// TIA Portal V14 SP1 export
// export: Created 2019-05-16T13:33:21.7383868Z, ExportSetting WithDefaults, WithReadOnly, DisplayName Totally Integrated Automation Portal, DisplayVersion V14 SP1 Update 6, DisplayName TIA Portal Openness, DisplayVersion V14 SP1 Update 6, DisplayName STEP 7 Professional, DisplayVersion V14 SP1 Update 6, DisplayName WinCC Professional, DisplayVersion V14 SP1 Update 6
FUNCTION_BLOCK "408М_Компрессор"   // FB2026, LAD
{ S7_Optimized_Access := 'FALSE' }
VERSION : 0.1
// stored: AutoNumber false, CodeModifiedDate 2019-03-26T07:08:54.9645568Z, CompileDate 2019-03-26T07:08:54.9928771Z, CreationDate 2019-02-26T05:18:41.6523018Z, InterfaceModifiedDate 2019-03-06T13:28:02.3471097Z, IsConsistent true, IsIECCheckEnabled false, IsKnowHowProtected false, ISMultiInstanceCapable true, IsWriteProtected false, LibraryConformanceStatus Warning: The object contains access to global data blocks. Warning: The block contains direct access to inputs, outputs, bit memories, indirect access to the registry or indirect access to external memory areas that are unknown at the time of compilation., ModifiedDate 2019-03-26T07:08:54.9645568Z, ParameterModified 2019-01-09T12:59:30.7163193Z, StructureModified 2019-03-06T13:28:02.3471097Z, UDAEnableTagReadback false
   VAR DB_SPECIFIC
      HMI : Struct
         CMD : Struct
            Start : Bool;   // Команда старта вибратора
            Stop : Bool;   // Команда останова вибратора
            Spare_2 : Bool;
            Spare_3 : Bool;
            Spare_4 : Bool;
            Spare_5 : Bool;
            Manual : Bool;
            Reset_Error : Bool;   // Сброс ошибок
         END_STRUCT;
         DATA : Struct
            StatusWord : Word;
            CntFbkTime : DInt := 4;   // Время контроля включения реле
            TimeDelay_SP : DInt := 2;   // Задержка срабатывания датчика давления
            Rot_Off_Time : Int;   // Обратный отсчет времени задержки запуска
            Line_Pressure_OK : Bool;   // Датчик давления компрессора ОК / Датчик давления в линии компрессора ОК
            Compressor_Pressure_OK : Bool;   // Датчик давления компрессора ОК
            Spare_7 : Bool;
            Spare_8 : Bool;
            Spare_9 : Bool;
            Spare_10 : Bool;
            Spare_11 : Bool;
            Spare_6 : Bool;
            Line_Presure : Real;   // Значение давления в линии
         END_STRUCT;
      END_STRUCT;
   END_VAR
   VAR
      One_Motor : "OneMotorManag";
      TOF : TOF;
      TOF_1 : TOF;
      TP : TP;
   END_VAR
   VAR DB_SPECIFIC
      CntFbkTime : Time;
      TimeDelay_SP : Time;
      StopTime : Time;   // Время остановки мотора компрессора
      Line_Presure : Real;   // Значение давления в линии
      Sensor_SP_OK : Bool;   // Датчик давления OK
      ResetErr : Bool;   // Сброс ошибок / Dumping of errors of the control package
      General_cond_OK : Bool;   // Готовность электрических систем / Conditions of permission of operation of the mechanism are not satisfied
      ManCmd_StartMov : Bool;   // Старт вращения в ручном режиме / Existence of command for rotation of the motor in manual
      ManCmd_StopMov : Bool;   // Стоп вращения в ручном режиме / Existence of command for a stop of rotation of the motor in manual
      AutoCmd_StartMov : Bool;   // Старт вращения в автоматическом режиме / Existence of command for rotation of the motor in the automatic
      AutoCmd_StopMov : Bool;   // Стоп вращения в автоматическом режиме / Existence of command for a stop of rotation of the motor in the automatic
   END_VAR
   VAR_TEMP
      FErr : Bool;   // Command 1 on operation of the mechanism in the automatic mode
      Temp_DINT : DInt;
   END_VAR
   VAR_TEMP   // added for the SCL form of the ladder/FBD networks
      _w1 : Bool;
      _w2 : Bool;
   END_VAR
BEGIN

REGION Network 2: Сброс ошибок
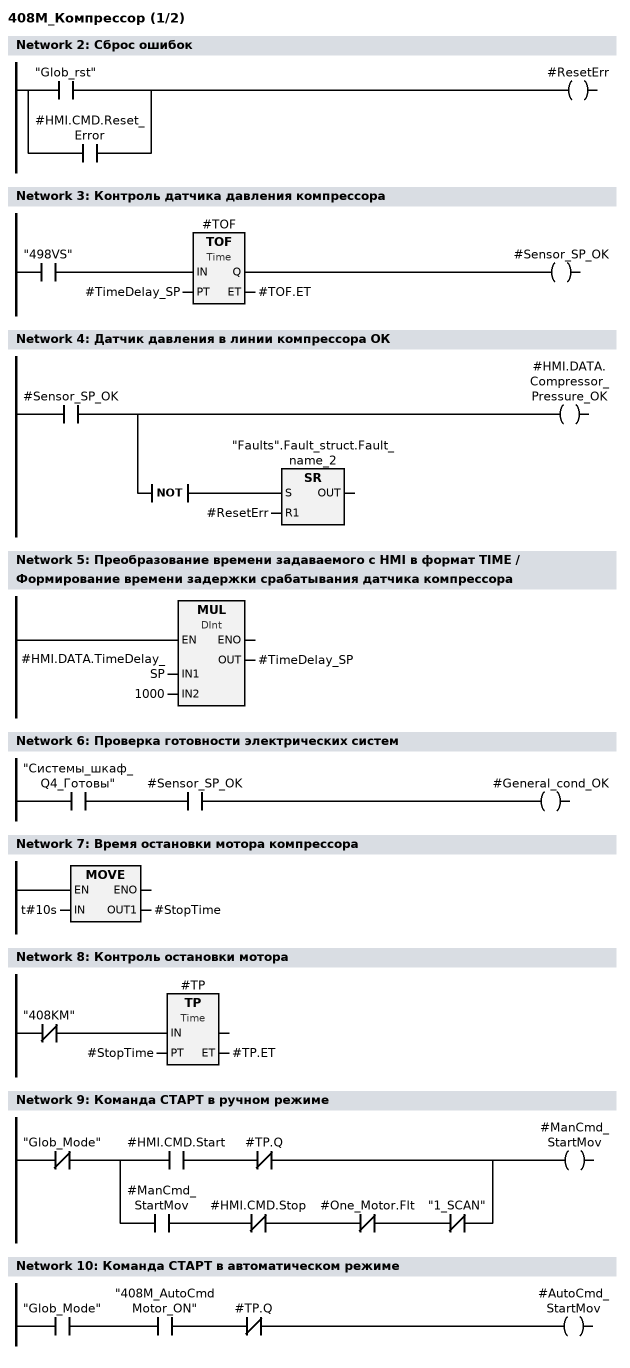
   RUNG wire#powerrail
      Contact( "Glob_rst" )
      wire#w1
      Coil( #ResetErr )
   END_RUNG
   RUNG wire#powerrail
      Contact( #HMI.CMD.Reset_Error )
   END_RUNG wire#w1
   // the same network as SCL:
   #ResetErr := "Glob_rst" OR #HMI.CMD.Reset_Error;
END_REGION

REGION Network 3: Контроль датчика давления компрессора
   RUNG wire#powerrail
      Contact( "498VS" )
      { S7_Templates := "time_type := Time" } #TOF.TOF(pt := #TimeDelay_SP, et => #TOF.ET)
      Coil( #Sensor_SP_OK )
   END_RUNG
   // the same network as SCL:
   #TOF.TOF(IN := "498VS", PT := #TimeDelay_SP, ET => #TOF.ET);
   #Sensor_SP_OK := #TOF.Q;
END_REGION

REGION Network 4: Датчик давления в линии компрессора ОК
   RUNG wire#powerrail
      Contact( #Sensor_SP_OK )
      wire#w1
      Coil( #HMI.DATA.Compressor_Pressure_OK )
   END_RUNG
   RUNG wire#w1
      Not()
      S_SR(operand := "Faults".Fault_struct.Fault_name_2, r1 := #ResetErr)
   END_RUNG
   // the same network as SCL:
   #HMI.DATA.Compressor_Pressure_OK := #Sensor_SP_OK;
   IF NOT #Sensor_SP_OK THEN
       "Faults".Fault_struct.Fault_name_2 := TRUE;   // SR flip-flop
   END_IF;
   IF #ResetErr THEN "Faults".Fault_struct.Fault_name_2 := FALSE; END_IF;
END_REGION

REGION Network 5: Преобразование времени задаваемого с HMI в формат TIME / Формирование времени задержки срабатывания датчика компрессора
   RUNG wire#powerrail
      { S7_Templates := "SrcType := DInt"; S7_GenerateENO := "TRUE" } Mul(in1 := #HMI.DATA.TimeDelay_SP, in2 := 1000, out => #TimeDelay_SP)
   END_RUNG
   // the same network as SCL:
   #TimeDelay_SP := #HMI.DATA.TimeDelay_SP * 1000;
END_REGION

REGION Network 6: Проверка готовности электрических систем
   RUNG wire#powerrail
      Contact( "Системы_шкаф_Q4_Готовы" )
      Contact( #Sensor_SP_OK )
      Coil( #General_cond_OK )
   END_RUNG
   // the same network as SCL:
   #General_cond_OK := "Системы_шкаф_Q4_Готовы" AND #Sensor_SP_OK;
END_REGION

REGION Network 7: Время остановки мотора компрессора
   RUNG wire#powerrail
      { S7_GenerateENO := "TRUE" } Move(in := t#10s, out1 => #StopTime)
   END_RUNG
   // the same network as SCL:
   #StopTime := t#10s;
END_REGION

REGION Network 8: Контроль остановки мотора
   RUNG wire#powerrail
      I_Contact( "408KM" )
      { S7_Templates := "time_type := Time" } #TP.TP(pt := #StopTime, et => #TP.ET)
   END_RUNG
   // the same network as SCL:
   #TP.TP(IN := NOT "408KM", PT := #StopTime, ET => #TP.ET);
END_REGION

REGION Network 9: Команда СТАРТ в ручном режиме
   RUNG wire#powerrail
      I_Contact( "Glob_Mode" )
      wire#w1
      Contact( #HMI.CMD.Start )
      I_Contact( #TP.Q )
      wire#w2
      Coil( #ManCmd_StartMov )
   END_RUNG
   RUNG wire#w1
      Contact( #ManCmd_StartMov )
      I_Contact( #HMI.CMD.Stop )
      I_Contact( #One_Motor.Flt )
      I_Contact( "1_SCAN" )
   END_RUNG wire#w2
   // the same network as SCL:
   #ManCmd_StartMov := NOT "Glob_Mode" AND ((#HMI.CMD.Start AND NOT #TP.Q) OR (#ManCmd_StartMov AND NOT #HMI.CMD.Stop AND NOT #One_Motor.Flt AND NOT "1_SCAN"));
END_REGION

REGION Network 10: Команда СТАРТ в автоматическом режиме
   RUNG wire#powerrail
      Contact( "Glob_Mode" )
      Contact( "408M_AutoCmdMotor_ON" )
      I_Contact( #TP.Q )
      Coil( #AutoCmd_StartMov )
   END_RUNG
   // the same network as SCL:
   #AutoCmd_StartMov := "Glob_Mode" AND "408M_AutoCmdMotor_ON" AND NOT #TP.Q;
END_REGION

REGION Network 11: Преобразование времени задаваемого с HMI в формат TIME
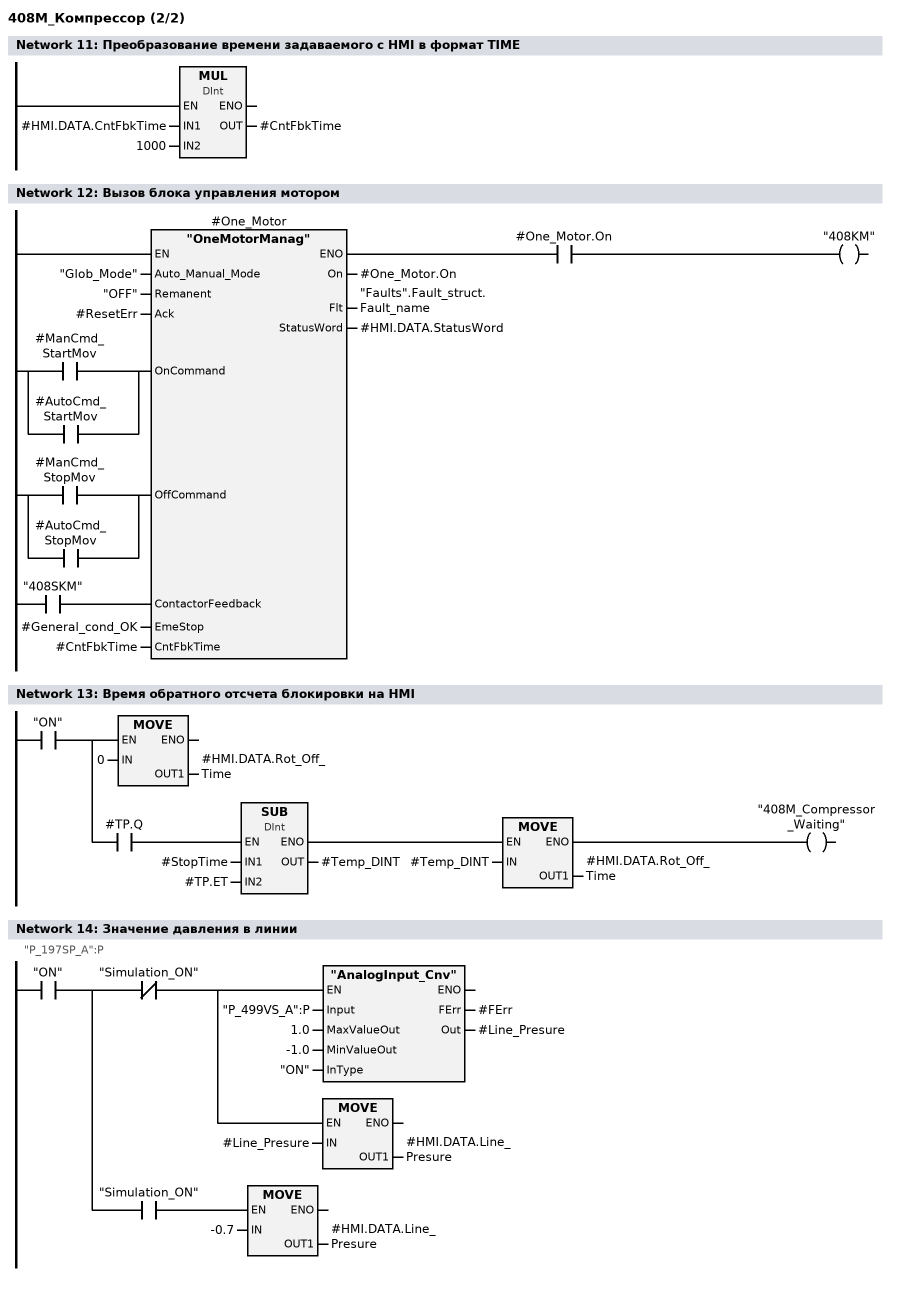
   RUNG wire#powerrail
      { S7_Templates := "SrcType := DInt"; S7_GenerateENO := "TRUE" } Mul(in1 := #HMI.DATA.CntFbkTime, in2 := 1000, out => #CntFbkTime)
   END_RUNG
   // the same network as SCL:
   #CntFbkTime := #HMI.DATA.CntFbkTime * 1000;
END_REGION

REGION Network 12: Вызов блока управления мотором
   RUNG wire#powerrail
      #One_Motor(OnCommand := wire#w1, OffCommand := wire#w2, ContactorFeedback := wire#w3, Auto_Manual_Mode := "Glob_Mode", Remanent := "OFF", Ack := #ResetErr, EmeStop := #General_cond_OK, CntFbkTime := #CntFbkTime, On => #One_Motor.On, Flt => "Faults".Fault_struct.Fault_name, StatusWord => #HMI.DATA.StatusWord)
      Contact( #One_Motor.On )
      Coil( "408KM" )
   END_RUNG
   RUNG wire#powerrail
      Contact( #ManCmd_StartMov )
   END_RUNG wire#w1
   RUNG wire#powerrail
      Contact( #AutoCmd_StartMov )
   END_RUNG wire#w1
   RUNG wire#powerrail
      Contact( #ManCmd_StopMov )
   END_RUNG wire#w2
   RUNG wire#powerrail
      Contact( #AutoCmd_StopMov )
   END_RUNG wire#w2
   RUNG wire#powerrail
      Contact( "408SKM" )
   END_RUNG wire#w3
   // the same network as SCL:
   #One_Motor(Auto_Manual_Mode := "Glob_Mode",   // "OneMotorManag"
              Remanent := "OFF",
              Ack := #ResetErr,
              OnCommand := #ManCmd_StartMov OR #AutoCmd_StartMov,
              OffCommand := #ManCmd_StopMov OR #AutoCmd_StopMov,
              ContactorFeedback := "408SKM",
              EmeStop := #General_cond_OK,
              CntFbkTime := #CntFbkTime,
              On => #One_Motor.On,
              Flt => "Faults".Fault_struct.Fault_name,
              StatusWord => #HMI.DATA.StatusWord,
              ENO => #_w1);
   "408KM" := #_w1 AND #One_Motor.On;
END_REGION

REGION Network 13: Время обратного отсчета блокировки на HMI
   RUNG wire#powerrail
      Contact( "ON" )
      wire#w1
      { S7_GenerateENO := "TRUE" } Move(in := 0, out1 => #HMI.DATA.Rot_Off_Time)
   END_RUNG
   RUNG wire#w1
      Contact( #TP.Q )
      { S7_Templates := "SrcType := DInt"; S7_GenerateENO := "TRUE" } Sub(in1 := #StopTime, in2 := #TP.ET, out => #Temp_DINT)
      { S7_GenerateENO := "TRUE" } Move(in := #Temp_DINT, out1 => #HMI.DATA.Rot_Off_Time)
      Coil( "408M_Compressor_Waiting" )
   END_RUNG
   // the same network as SCL:
   // ENO of a box is taken as its EN; it also drops when the box reports an error
   IF "ON" THEN #HMI.DATA.Rot_Off_Time := 0; END_IF;
   #_w1 := "ON" AND #TP.Q;
   IF #_w1 THEN
       #Temp_DINT := #StopTime - #TP.ET;
       #HMI.DATA.Rot_Off_Time := #Temp_DINT;
   END_IF;
   "408M_Compressor_Waiting" := #_w1;
END_REGION

REGION Network 14: Значение давления в линии
   // "P_197SP_A":P
   RUNG wire#powerrail
      Contact( "ON" )
      wire#w1
      I_Contact( "Simulation_ON" )
      wire#w2
      "AnalogInput_Cnv"(Input := "P_499VS_A":P, MaxValueOut := 1.0, MinValueOut := -1.0, InType := "ON", FErr => #FErr, Out => #Line_Presure)
   END_RUNG
   RUNG wire#w2
      { S7_GenerateENO := "TRUE" } Move(in := #Line_Presure, out1 => #HMI.DATA.Line_Presure)
   END_RUNG
   RUNG wire#w1
      Contact( "Simulation_ON" )
      { S7_GenerateENO := "TRUE" } Move(in := -0.7, out1 => #HMI.DATA.Line_Presure)
   END_RUNG
   // the same network as SCL:
   #_w1 := "ON";
   #_w2 := "ON" AND NOT "Simulation_ON";
   IF #_w2 THEN
       "AnalogInput_Cnv"(Input := "P_499VS_A":P,
                         MaxValueOut := 1.0,
                         MinValueOut := -1.0,
                         InType := "ON",
                         FErr => #FErr,
                         Out => #Line_Presure);
       #HMI.DATA.Line_Presure := #Line_Presure;
   END_IF;
   IF #_w1 AND "Simulation_ON" THEN #HMI.DATA.Line_Presure := -0.7; END_IF;
END_REGION
END_FUNCTION_BLOCK
